{attribute 'OPC.UA.DA.StructuredType' := '1'}
FUNCTION_BLOCK FB_Unit_RO_PW30_1 EXTENDS FB_BaseDevice IMPLEMENTS I_Device

VAR
	{attribute 'OPC.UA.DA' := '1'} 
	bInContactor AT %I*: BOOL := FALSE;
	{attribute 'OPC.UA.DA' := '1'} 
	bInRun AT %I*: BOOL := FALSE;
	{attribute 'OPC.UA.DA' := '1'} 
	bInAlarm AT %I*: BOOL := FALSE;
	
	{attribute 'OPC.UA.DA' := '1'} 
	bOutContactor AT %Q*: BOOL := FALSE;
	{attribute 'OPC.UA.DA' := '1'} 
	bOutON AT %Q*: BOOL := FALSE;
	{attribute 'OPC.UA.DA' := '1'} 
	bOutEnable AT %Q*: BOOL := FALSE;
	
	{attribute 'OPC.UA.DA' := '0'} 
	eSMState: (WAIT, TURNING_ON, ON, TURNING_OFF, OFF);
	
	{attribute 'OPC.UA.DA' := '0'} 
	tActionTimeout: TIME := T#5S;
	{attribute 'OPC.UA.DA' := '0'} 
	fbTON_timeout: TON := (PT := tActionTimeout, IN := FALSE);
END_VAR

fbTONstartTime();
fbTONstopTime();

IF GVL.bAutoUpdateDeviceState THEN
	eState := eStateTarget;	
END_IF


IF bEnable THEN
	IF eStateTarget = E_DeviceState.ON AND eState <> E_DeviceState.ON THEN
		eSMState := TURNING_ON;
	END_IF
END_IF

IF eStateTarget = E_DeviceState.OFF AND eState <> E_DeviceState.OFF THEN
		eSMState := TURNING_OFF;
END_IF

IF bInAlarm THEN
	raiseAlarm(Priority := E_AlarmPriority.High, Label := 'Unit Alarm Active', Enabled := TRUE, DeviceAlarmID := 1);
END_IF


CASE eSMState OF
	
	WAIT:
		//Wait for method call to change ESMState
		
	TURNING_ON: 
		eState := E_DeviceState.TURNING_ON;
		
		bOutContactor := TRUE;
		bOutEnable := TRUE;
		bOutON := TRUE;
	
		
		IF fbTONstartTime.Q THEN
			eSMState := WAIT;
			raiseAlarm(Priority := E_AlarmPriority.High, Label := 'Failed to Start', Enabled := TRUE, DeviceAlarmID := 2);
		END_IF
		
		IF bInContactor AND bInRun THEN
			eSMState := ON;
			eState := E_DeviceState.ON;
		END_IF
		
	ON:
		IF bInContactor <> TRUE THEN
			raiseAlarm(Priority := E_AlarmPriority.High, Label := 'Power Lost', Enabled := TRUE, DeviceAlarmID := 1);
			eState := E_DeviceState.OFF;
			eSMState := WAIT;
		END_IF
		
		IF bInRun <> TRUE THEN
			raiseAlarm(Priority := E_AlarmPriority.High, Label := 'Unit Stopped Running', Enabled := TRUE, DeviceAlarmID := 2);
			eState := E_DeviceState.OFF;
			eSMState := WAIT;
		END_IF
			
		
	TURNING_OFF:
		eState := E_DeviceState.TURNING_OFF;
		bOutContactor := FALSE;
		bOutON := FALSE;
		bOutEnable := FALSE;
				
		IF fbTONstopTime.Q THEN
			eSMState := WAIT;
			raiseAlarm(Priority := E_AlarmPriority.High, Label := 'Failed to Stop', Enabled := TRUE, DeviceAlarmID := 3);
		END_IF 
		
		IF bInRun = FALSE AND bInContactor = FALSE THEN
			eSMState := OFF;	
		END_IF
		

	OFF:
		eState := E_DeviceState.OFF;
		eSMState := WAIT;
		
		
END_CASE

{warning 'add method implementation '}
METHOD disable : BOOL
bEnable := FALSE;
END_METHOD

{warning 'add method implementation '}
METHOD enable : BOOL
bEnable := TRUE;
END_METHOD

METHOD FB_init : BOOL
VAR_INPUT
	bInitRetains : BOOL; // if TRUE, the retain variables are initialized (warm start / cold start)
	bInCopyCode : BOOL;  // if TRUE, the instance afterwards gets moved into the copy code (online change)
	
	UnitID: STRING(80);
	UnitDescr: STRING(255); 
END_VAR
sID := UnitID;
sDescr := UnitDescr;
END_METHOD

METHOD setOff : BOOL
VAR_INPUT
END_VAR
eSMState := TURNING_OFF;
END_METHOD

METHOD setOn : BOOL
VAR_INPUT
END_VAR
eSMState := TURNING_ON;
END_METHOD

END_FUNCTION_BLOCK

(* stored: Version 1.1.0.1, ProductVersion 3.1.4024.12
   POU FB_Unit_RO_PW30_1: Id {83f55630-35da-4827-a34e-80f23b0d6314}, SpecialFunc None
   Method disable: Id {de9b2d5e-8374-44c3-9afa-d4f1a13118e6}
   Method enable: Id {95c83e89-77dc-486f-b190-f06a1328fe43}
   Method FB_init: Id {4c919149-38b0-43f4-8c9e-3b5f7939d240}
   Method setOff: Id {2bf024f8-ee2e-4156-8032-230eeb4b46a6}
   Method setOn: Id {5171bf36-8220-402d-b2c7-b945102013e4} *)
